// TIA Portal V19 export
TYPE "Analogic_SensorManagement_Par"
// stored: Access Published
   STRUCT
      Enable : Bool;
      RangeLow : Real;
      RangeHigh : Real;
   END_STRUCT;
END_TYPE
